TYPE ST_Data :
STRUCT
	viewer	: ST_Viewer;
END_STRUCT
END_TYPE

(* stored: Version 1.1.0.1, ProductVersion 3.1.4024.11
   DUT ST_Data: Id {3df07c4d-8e31-4786-8513-6e99693c4b11} *)
